FUNCTION_BLOCK FB_Ampel
VAR_INPUT
	estate : eBetriebszustand;
END_VAR
VAR_OUTPUT
	bAmpelgruen : BOOL;
	bAmpelrot : BOOL;
	bAmpelgelb : BOOL;
END_VAR
VAR
	Ampel_blinken : FB_Blinklicht;
END_VAR

//Die Ampel leuchtet je nach Betriebszustand in unterschiedlichen Farben, um diesen anzuzeigen
CASE estate OF
	
	eBetriebszustand.off:
	bAmpelgruen := FALSE;
	bAmpelrot := TRUE;
	bAmpelgelb := FALSE;	
	
	eBetriebszustand.init:
	bAmpelrot := FALSE;
	bAmpelgelb := FALSE;
	Ampel_blinken(bStartStop:=TRUE , tPeriode:= , bBlink=>bAmpelgruen );
	
	eBetriebszustand.ready:
	bAmpelrot := FALSE;
	Ampel_blinken(bStartStop:=TRUE , tPeriode:= , bBlink=>bAmpelgelb );
	bAmpelgruen := NOT bAmpelgelb;
	//gruen_blinken(bStartStop:=True , tPeriode:= , bBlink=>bAmpelgruen );
	
	eBetriebszustand.production:
	bAmpelrot := FALSE;
	bAmpelgelb := FALSE;
	bAmpelgruen := TRUE;
	
	eBetriebszustand.done:
	bAmpelgruen := TRUE;
	bAmpelrot := FALSE;
	bAmpelgelb := TRUE;	
	
END_CASE

END_FUNCTION_BLOCK

(* stored: Version 1.1.0.1, ProductVersion 3.1.4024.15
   POU FB_Ampel: Id {26ef8762-be59-4741-8ba7-897e4ca54110}, SpecialFunc None *)
